// TIA Portal V17 export
// export: Created 2022-02-03T14:45:11.6470527Z, ExportSetting WithDefaults, DisplayName Totally Integrated Automation Portal, DisplayVersion V17, DisplayName TIA Portal Openness, DisplayVersion V17, DisplayName TIA Portal Version Control Interface, DisplayVersion V17, DisplayName SINAMICS Startdrive Advanced, DisplayVersion V17, DisplayName SINAMICS Startdrive G130, G150, S120, S150, SINAMICS MV, S210, DisplayVersion V17, DisplayName SINAMICS Startdrive G110M, G120, G120C, G120D, G120P, G115D, DisplayVersion V17, DisplayName STEP 7 Professional, DisplayVersion V17, DisplayName STEP 7 Safety, DisplayVersion V17, DisplayName WinCC Advanced, DisplayVersion V17
FUNCTION "SignalBay" : Bool   // FC3, LAD
VERSION : 0.1
// stored: Access Published, AutoNumber true, IsIECCheckEnabled false, SetENOAutomatically false, UDAEnableTagReadback false
   VAR_INPUT
      operation : Bool;   // Operation mode
      bBay : Bool;   // sensor bay x
      sBay : Bool;   // Momentary contact bay x
      occupiedBay : Bool;   // Bay occupied
      frequ2Hz : Bool;   // 2Hz frequency
   END_VAR
   // Ret_Val : LED bay x
BEGIN

REGION Network 1: LED bay x
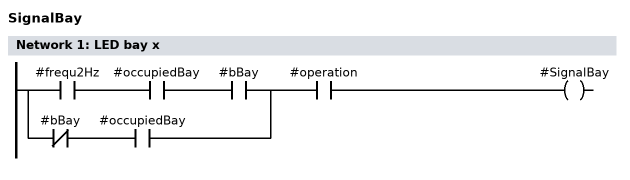
   RUNG wire#powerrail
      Contact( #frequ2Hz )
      Contact( #occupiedBay )
      Contact( #bBay )
      wire#w1
      Contact( #operation )
      Coil( #SignalBay )
   END_RUNG
   RUNG wire#powerrail
      I_Contact( #bBay )
      Contact( #occupiedBay )
   END_RUNG wire#w1
   // the same network as SCL:
   #SignalBay := ((#frequ2Hz AND #occupiedBay AND #bBay) OR (NOT #bBay AND #occupiedBay)) AND #operation;
END_REGION
END_FUNCTION
